{attribute 'GeneratedUsingTerminal: AT2050-0501-0024'}
{attribute addProperty BoxType "AT2050-0501-0024"}
{attribute addProperty Id "A_0084_AT2050_5500_0017_AT2050_5500AT2050_33A3DF1B80"}
{attribute addProperty CRC "99014176"}
{attribute addProperty Size "80"}
TYPE A_0072_AT2050_0501_0024_AT2050_0501_05E6D620 EXTENDS AT2050_2EA6C9BF :
STRUCT
	{attribute addProperty Name "A_0084_AT2050_5500_0017_AT2050_5500"}
	{attribute addProperty PreviousPort "A_0072(AT2050-0501-0024) (AT2050-0501) : B"}
	A_0084_AT2050_5500_0017_AT2050_5500 : AT2050_33A3DF1B;
END_STRUCT
END_TYPE

(* stored: Version 1.2.0.0, ProductVersion 3.1.4024.9
   DUT A_0072_AT2050_0501_0024_AT2050_0501_05E6D620: Id {6c172824-ad5c-4539-be7f-116c9df8c797} *)
